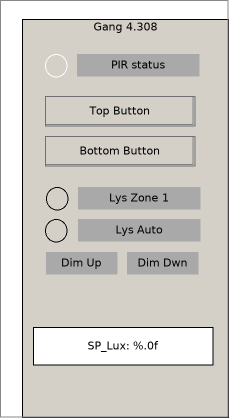
VISUALIZATION Visualization_4_308_1_1  // 229x418
    RoundedRectangle (22,19 207x399), "Gang 4.308"
    Rectangle (33,327 180x38), "SP_Lux: %.0f", text variable: P_Gang_4_308.arrfbLysGruppe[1].fbLightCtrl.fLuxZone1
    Button (45,96 150x30), "Top Button"
        tap P_Gang_4_308.bButtonZone1_Visu
    Button (45,136 150x30), "Bottom Button"
        tap P_Gang_4_308.bBottomButtonZone1_Visu
    Ellipse (46,187 22x23), colour toggle: P_Gang_4_308.fbLys.fbLightCtrl.bOnZone1
    Rectangle (78,187 122x22), "Lys Zone 1"
    Rectangle (46,252 71x22), "Dim Up", colour toggle: P_Gang_4_308.arrfbLysGruppe[1].fbLightCtrl.bDimUp
    Rectangle (127,252 71x22), "Dim Dwn", colour toggle: P_Gang_4_308.arrfbLysGruppe[1].fbLightCtrl.bDimDwn
    Ellipse (45,219 22x23), colour toggle: P_Gang_4_308.arrfbLysGruppe[1].fbLightCtrl.bAutoZone1
    Rectangle (78,219 122x22), "Lys Auto"
    Ellipse (45,54 22x23), colour toggle: P_Gang_4_308.arrfbLysGruppe[1].fbLightCtrl.bPIR
    Rectangle (77,54 122x22), "PIR status"
END_VISUALIZATION

(* stored: Version 1.1.0.1
   Visu Visualization_4_308_1_1: Id {40992399-fedf-46ba-9240-72ce2092f435} *)
